(* PLC project Unnamed, Unknown Unnamed 1 *)
(* stored: creationDateTime 2021-08-03T19:17:13, modificationDateTime 2021-08-04T17:47:23 *)

(* x100 *)
PROGRAM program0
  VAR
    X100 : BOOL;
    X101 : BOOL;
    Y100 : BOOL;
  END_VAR

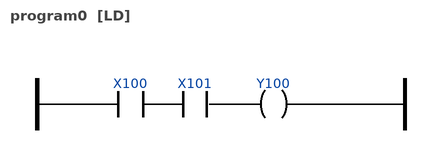
(* LD diagram, written out as Structured Text *)
Y100 := X100 AND X101;
END_PROGRAM

CONFIGURATION Config0
  RESOURCE Res0 ON PLC
    TASK task0(INTERVAL := T#20ms, PRIORITY := 0);
    PROGRAM instance0 WITH task0 : program0;
  END_RESOURCE
END_CONFIGURATION
